TYPE DUT_SensorHGS:
STRUCT
    fCntsInEGU:			REAL;
    {attribute 'pytmc' := '
        pv: EU
        io: i
    '}
    sEGU:				STRING;
    sName:				STRING;
    {attribute 'pytmc' := '
        pv: VALUE
        io: i
    '}
    fValue:				REAL;
    {attribute 'pytmc' := '
        pv: RAWCOUNTS
        io: i
    '}
    iRawCnts AT %I*:	DINT;
    iOffset:			DINT;
END_STRUCT
END_TYPE

(* stored: Version 1.1.0.1
   DUT DUT_SensorHGS: Id {2917fbec-0023-49ad-b5e9-7d9d5133fd10} *)
